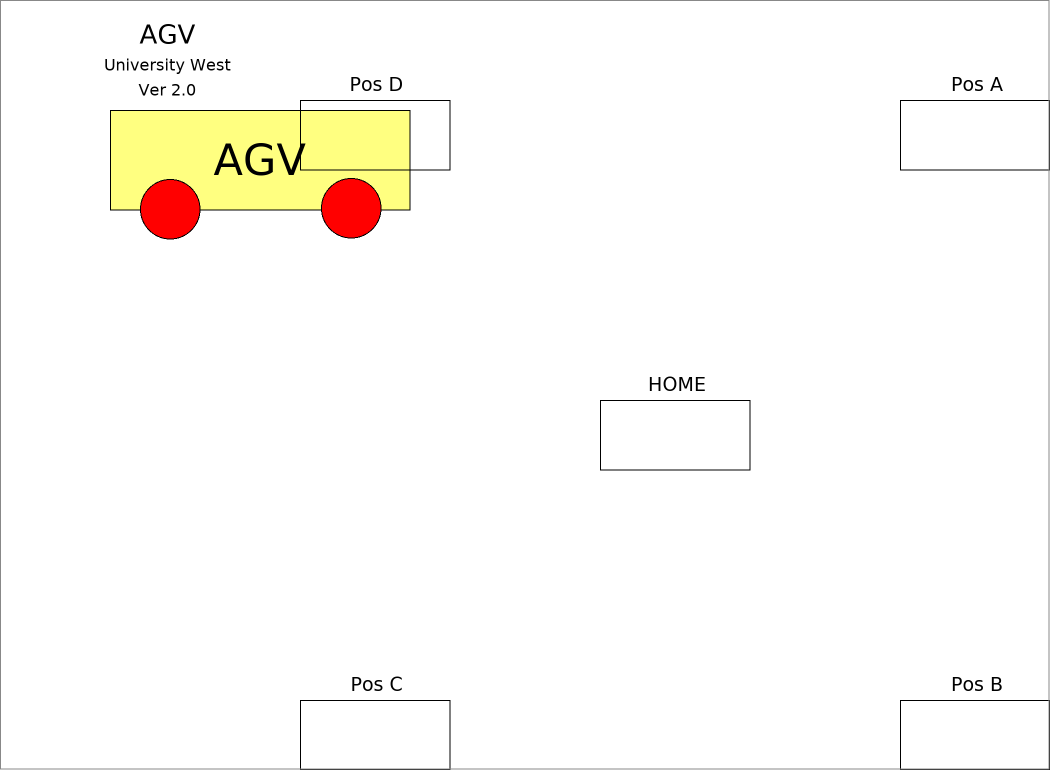
VISUALIZATION AGVSimulator  // 1050x770
    Group (110,110 130x50)
        p3560616238: Process.fbAGV.iAtPos_X
        p2738717112: Process.fbAGV.iAtPos_Y
        RoundedRectangle (0,0 300x100), "AGV"
        Ellipse (30,69 60x60)
        Ellipse (211,68 60x60)
    RoundedRectangle (300,100 150x70)
    RoundedRectangle (900,100 150x70)
    RoundedRectangle (600,400 150x70)
    RoundedRectangle (900,700 150x70)
    RoundedRectangle (300,700 150x70)
    Rectangle (330,670 94x29), "Pos C"
    Rectangle (930,670 94x29), "Pos B"
    Rectangle (930,70 94x29), "Pos A"
    Rectangle (330,70 93x29), "Pos D"
    Rectangle (630,370 94x29), "HOME"
    Rectangle (130,370 94x29), "ERROR", invisible if: NOT Process.fbAGV.xError
    Rectangle (80,20 175x29), "AGV"
    Rectangle (80,50 175x30), "University West"
    Rectangle (80,75 175x30), "Ver 2.0"
    RoundedRectangle (107,356 144x54), invisible if: Process.fbAGV.xError
END_VISUALIZATION

(* stored: Version 1.1.0.1
   Visu AGVSimulator: Id {5384fcf8-819a-41bf-bdf0-d486f0b6248b} *)
